Staubli VAL3: stop.pgx

program stop()
begin

  stopMove()
  resetMotion()
  disablePower()
  userPage("new1")
  call cakajProgress(2)
end
